DATA_BLOCK "bioSig.DB"
{ S7_Optimized_Access := 'TRUE' }
VERSION : 1.0
// Batch I/O Sig Data Block:
// by Woermann Automation
NON_RETAIN
   VAR RETAIN
      sig : Array[0..15] of "bioSig.DT";
   END_VAR

BEGIN

END_DATA_BLOCK

